Universal Robots PolyScope program: one_urcap.urp

Program one_urcap (installation=default directory=/ursim/programs createdIn=5.11.1.108318 lastSavedIn=5.11.1.108318 robotSerialNumber=20195599999)
Calibrated DH parameters: a=[0, -0.425, -0.3922, 0, 0, 0]; d=[0.1625, 0, 0, 0.1333, 0.0997, 0.0996]; alpha=[1.570796, 0, 0, 1.570796, -1.570796, 0]; deltaTheta=[0, 0, 0, 0, 0, 0]
Robot Program (runOnlyOnce=true)
  Wait Sleep waitTime=1
  URCap External Control (External Control, FZI Research Center for Information Technology)
